FUNCTION_BLOCK EV_MERGE (* Composite Function Block Type *)
  (* Standard: 61499-2 *)
  (* Version 0.0, 2/9/2018, Sandeep Patil, nxtControl GmbH, template *)
  PACKAGE Main;
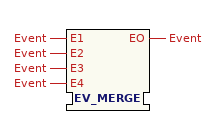
  EVENT_INPUT
    E1; (* Initialization Request *)
    E2; (* Normal Execution Request *)
    E3;
    E4;
  END_EVENT
  EVENT_OUTPUT
    EO; (* Initialization Confirm *)
  END_EVENT
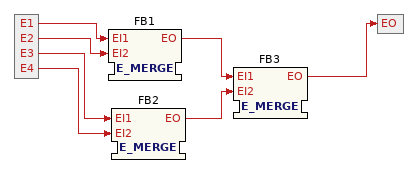
  FBS
    FB1 : E_MERGE;
    FB2 : E_MERGE;
    FB3 : E_MERGE;
  END_FBS
  EVENT_CONNECTIONS
    E1 TO FB1.EI1;
    E2 TO FB1.EI2;
    E3 TO FB2.EI1;
    E4 TO FB2.EI2;
    FB1.EO TO FB3.EI1;
    FB2.EO TO FB3.EI2;
    FB3.EO TO EO;
  END_CONNECTIONS
END_FUNCTION_BLOCK
